FUNCTION_BLOCK FB_PIZZA_OVEN 
VAR_INPUT
	Pizza_in 	: 			BOOL:=FALSE;
	Pizza_out 	:			BOOL:=FALSE;

	fbTrig		: 			R_TRIG;
	fbTrig2		: 			R_TRIG;
END_VAR

VAR_OUTPUT
	PizzaStatus	: 			STRING;
END_VAR
VAR
	_pizza_aus: 			BOOL;
	_pizza_ein:				BOOL;
	_brand_alarm: 			BOOL;
	_cook_time:				TIME;
		_count	:			DINT;
	
	fbTimer		: 			TON;
	fbTimer1	:			TON;
	
	_pizza_backen:			BOOL;
	
	_teig_auflade:			BOOL;

	_zutaten		:		BOOL;

	_pizza_fertig:			BOOL;
	_led_anzeige:			BOOL;

	iState		:  			DINT:=0;
	
END_VAR

PROPERTY BrandAlarm : BOOL
GET
BrandAlarm:=_brand_alarm;
END_GET
SET
_brand_alarm:=BrandAlarm;
END_SET
END_PROPERTY

PROPERTY IngridientDeck : BOOL
GET
IngridientDeck:=_zutaten;
END_GET
SET
_zutaten:=IngridientDeck;
END_SET
END_PROPERTY

PROPERTY KochZeit : TIME
GET
KochZeit:=_cook_time;
END_GET
SET
_cook_time:=KochZeit;
END_SET
END_PROPERTY

PROPERTY LedAnzeige : BOOL
GET
LedAnzeige:= _led_anzeige;
END_GET
SET
_led_anzeige:= LedAnzeige;
END_SET
END_PROPERTY

METHOD MethodBrandAlarm : BOOL
VAR_INPUT
END_VAR
END_METHOD

METHOD MethodCounter : DINT
VAR_INPUT
END_VAR
_count:=_count+1;
END_METHOD

METHOD MethodLedAnzeige : BOOL
VAR_INPUT
END_VAR

_led_anzeige:=TRUE;
END_METHOD

METHOD PUBLIC MethodPizza : UDINT
VAR


END_VAR
//control buttons
THIS^.MethodPizzaAufladen();
THIS^.MethodRemovePizza();
//status changes
CASE iState OF 
0:	PizzaStatus:='Offen Frei';
IF _teig_auflade AND NOT _zutaten THEN		
		_teig_auflade:=FALSE;
		_zutaten:=TRUE;
END_IF
fbTimer1(IN:=_zutaten,PT:=T#3S);
IF fbTimer1.Q THEN
	iState:=7;
END_IF 	
7: IF _zutaten AND NOT _pizza_backen THEN
					
		_zutaten:=FALSE;
		_pizza_backen:=TRUE;
		iState:=10;
END_IF
10:	IF _pizza_backen THEN
	  PizzaStatus:='Öffen besetzt...';
	THIS^.MethodLedAnzeige();
END_IF
	fbTimer(IN:=_pizza_backen,PT:=KochZeit);
IF fbTimer.Q THEN
	//PizzaInOven:=FALSE;
	THIS^.MethodCounter();
	iState:=20;
	
END_IF
	
20:	PizzaStatus:='Entladen';
IF  NOT _pizza_fertig THEN
	_brand_alarm:=FALSE;
	_pizza_backen:=FALSE;
	_pizza_fertig:=TRUE;
	fbTimer(IN:=FALSE);
	iState:=0;
	ELSE
		_brand_alarm:=TRUE;
	END_IF
	
END_CASE
END_METHOD

METHOD MethodPizzaAufladen : BOOL
VAR_INPUT
END_VAR
		fbTrig(CLK:=_pizza_ein);//load pizza button clicked trggered
IF		fbTrig.Q THEN		//When Triggerd 
		_teig_auflade:=TRUE;	
			iState:=0;
		//Pizza_in:=FALSE;
		//fbTrig(clk:=FALSE);
END_IF
END_METHOD

METHOD MethodRemovePizza : BOOL
VAR_INPUT
END_VAR
	fbTrig2(CLK:=_pizza_aus); 
IF 	fbTrig2.Q THEN
	_pizza_fertig:=FALSE;
	//Pizza_out:=FALSE;
	//fbTrig2(clk:=Pizza_out);
END_IF
END_METHOD

PROPERTY PizzaAus : BOOL
GET
PizzaAus:=_pizza_aus;
END_GET
SET
_pizza_aus:=PizzaAus;
END_SET
END_PROPERTY

PROPERTY PizzaDone : BOOL
GET
PizzaDone:=_pizza_fertig;
END_GET
SET
_pizza_fertig:=PizzaDone;
END_SET
END_PROPERTY

PROPERTY PizzaEin : BOOL
GET
PizzaEin:=_pizza_ein;
END_GET
SET
_pizza_ein:=PizzaEin;
END_SET
END_PROPERTY

PROPERTY PizzaInOven : BOOL
GET
PizzaInOven:=_pizza_backen;
END_GET
SET
_pizza_backen:=PizzaInOven;
END_SET
END_PROPERTY

PROPERTY PizzaOnDeck : BOOL
GET
PizzaOnDeck:=_teig_auflade;
END_GET
SET
_teig_auflade:=PizzaOnDeck;
END_SET
END_PROPERTY

PROPERTY Zaehler : DINT
GET
Zaehler:=_count;
END_GET
SET
_count:=Zaehler;
END_SET
END_PROPERTY

END_FUNCTION_BLOCK

(* stored: Version 1.1.0.1, ProductVersion 3.1.4022.6
   POU FB_PIZZA_OVEN: Id {e54d8141-8c6a-4975-af63-b1ccd7a5bba4}, SpecialFunc None
   Property BrandAlarm: Id {f46e6aa1-263d-4a69-9523-9496ad1a28b8}
   Get Get: Id {38e0107e-4d2f-4a51-b202-875d8ce5ebc6}
   Set Set: Id {b5a5cd8e-ac06-4fea-8eda-d1f228cb77c6}
   Property IngridientDeck: Id {ea4e0c9b-9f8e-4059-91ce-d2642ed67783}
   Get Get: Id {8f289bdc-e694-425d-bf5e-5bf9c7822329}
   Set Set: Id {5d493b73-7a1f-4f56-9e55-1d0c622f8c60}
   Property KochZeit: Id {160a7534-386d-427b-b5aa-18f1f8198e2f}
   Get Get: Id {62fa3185-dfe5-4cd9-b957-7eb0d8e55629}
   Set Set: Id {6d1c1e6c-34a8-4e5e-9306-029957c80666}
   Property LedAnzeige: Id {4b30958b-1325-47fa-82c2-2c6b5a056ebd}
   Get Get: Id {8ca948e6-6c58-449b-9704-53c0d7cd339a}
   Set Set: Id {e16658f1-00c7-4723-8f39-aba3b2ac8a02}
   Method MethodBrandAlarm: Id {2acef4a8-b76f-4990-95c7-9507d2e4951d}
   Method MethodCounter: Id {4b44d077-033b-4f7e-a518-c3de8b5fa58c}
   Method MethodLedAnzeige: Id {ef754064-e191-49c6-a794-270d7cff6354}
   Method MethodPizza: Id {973a8685-4554-4338-ac21-4d340b906904}
   Method MethodPizzaAufladen: Id {41b55cfc-d288-41c3-9fdc-443befab6b0f}
   Method MethodRemovePizza: Id {2b4dedaf-8eb2-406a-a5bc-d1bccf5caf5e}
   Property PizzaAus: Id {93c4c040-ee33-4a6c-8279-1d3c3ab97d9f}
   Get Get: Id {7d6407b2-7a50-4242-9255-b2ce80bba508}
   Set Set: Id {af536bfb-2415-465b-8198-0980b8d9d50d}
   Property PizzaDone: Id {4f2739fa-260b-4ae1-acee-b971e5e03f1e}
   Get Get: Id {db4cf35a-1689-48af-8094-928878353f4a}
   Set Set: Id {ead687ea-5438-4bea-919f-24f6e4d82ddb}
   Property PizzaEin: Id {18d4b099-bcef-4881-acb4-0297dd08bd27}
   Get Get: Id {1a334dcc-9af8-4421-af00-f0501ca42bcc}
   Set Set: Id {9c7b20e6-744a-4c96-958d-42aa4a630643}
   Property PizzaInOven: Id {ee446f2d-cb89-4304-b383-b906b2f5a834}
   Get Get: Id {bab41a42-581d-4d13-b068-3c5f3f2690a8}
   Set Set: Id {d8e8d256-ef42-44bb-9d55-c21a05537254}
   Property PizzaOnDeck: Id {0c654e1e-b969-4063-a2d1-a8b1e9d8f7f0}
   Get Get: Id {779b6387-867b-48b4-997c-ed4ed0c5396e}
   Set Set: Id {5d90542b-3ef3-455e-b15d-b7cbc991d2eb}
   Property Zaehler: Id {0ff2f4b4-f3a8-4617-82b0-b7a068d35a6b}
   Get Get: Id {8d882e6f-35f8-4904-ab88-1ab5b2fe6ca5}
   Set Set: Id {e6f10d83-6106-43ee-88d9-73c3d242278d} *)
